Staubli VAL3: MoveLine.pgx

program MoveLine(num x_nX, num x_nY, num x_nZ, num x_nRx, num x_nRy, num x_nRz)
begin
  pPointRx.trsf.x = x_nX
  pPointRx.trsf.y = x_nY
  pPointRx.trsf.z = x_nZ
  pPointRx.trsf.rx = x_nRx
  pPointRx.trsf.ry = x_nRy
  pPointRx.trsf.rz = x_nRz
  movel(pPointRx,tCurrentTool,mCurrentSpeed)
end
